{attribute 'qualified_only'}
{attribute 'strict'}
{attribute 'to_string'}
TYPE ST145_Pnp_e :
(
    RESET := 0, // Reset

    INIT := 100, // Initialisieren 
    Init_HomeVerticals,
    Init_VerticalsUp,
    Init_HomeHorizontals,
    Init_HorizontalsToTrack,
    Init_check_if_pces_handled,

    MOVER_FREE_OP, // Ab here, operation without mover can be done
    READY := 999,  // READY to Start, Init Done 
    START := 1000, // Start Zyklisch

    PnP_Hor_ToRotTablePos,
    PnP_WaitOnFeeder,
    PnP_Ver_RotTableDown,
    Vacum_on,
    PnP_Ver_RotTableUp,
    PnP_Hor_ToTrackPos,
    waitOnMover,     // wait until the mover is there
    MOVER_NEEDED_OP, // Since here, a mover in position is needed to perform the action

    PnP_Ver_ShuttleDown,
    PnP_Ver_ShuttleTorqueControl,
    Vacum_off,
	Pnp_move_a_bit_to_feeder,
    PnP_Ver_ShuttleUp,

    SYNC_MOVER_LEAVE, // MoverMan need to take the mover
    DONE := 8000,     // Ablauf beendet 
    ERROR := 9000,    // Fehler 
    _max
);
END_TYPE

(* stored: Version 1.1.0.1, ProductVersion 3.1.4024.6
   EnumerationTextList ST145_Pnp_e: Id {69b8a2fa-26d6-4cd8-91cd-e4208d076d18} *)
